FUNCTION_BLOCK FB_HybridEnergyStorage
VAR_INPUT
END_VAR
VAR_OUTPUT
END_VAR
VAR
END_VAR

END_FUNCTION_BLOCK

(* stored: Version 1.1.0.1, ProductVersion 3.1.4024.10
   POU FB_HybridEnergyStorage: Id {d0e73ddc-d48c-401f-86b9-ea00e651427d}, SpecialFunc None *)
